// TIA Portal V17 export
// export: Created 2022-01-24T13:54:52.2363319Z, ExportSetting WithDefaults, DisplayName Totally Integrated Automation Portal, DisplayVersion V17 Update 1, DisplayName TIA Portal Openness, DisplayVersion V17 Update 1, DisplayName TIA Portal Teamcenter Gateway, DisplayVersion V17 Update 1, DisplayName TIA Portal Version Control Interface, DisplayVersion V17, DisplayName SINAMICS Startdrive Advanced, DisplayVersion V17 Update1, DisplayName SINAMICS Startdrive G110M, G120, G120C, G120D, G120P, G115D, DisplayVersion V17 Update1, DisplayName SINAMICS Startdrive G130, G150, S120, S150, SINAMICS MV, S210, DisplayVersion V17 Update1, DisplayName STEP 7 Professional, DisplayVersion V17 Update 1, DisplayName STEP 7 Safety, DisplayVersion V17, DisplayName Soft Starter ES, DisplayVersion V17, DisplayName WinCC Advanced, DisplayVersion V17 Update 1, DisplayName SIMATIC Visualization Architect, DisplayVersion V17
VAR_GLOBAL   // PLC tag table "Tag table_1"
   test01 AT %M101.0 : Bool;   //    {ExternalAccessible false, ExternalVisible false, ExternalWritable false}
END_VAR
